FUNCTION_BLOCK pidCtl (* Composite Function Block Type *)
  (* Standard: 61499-2 *)
  (* Version 1.0.1, 11/15/2023, ApplicationLibDevTeam, Schneider Electric, First Version *)
  PACKAGE Hidryco.HidrycoLib;
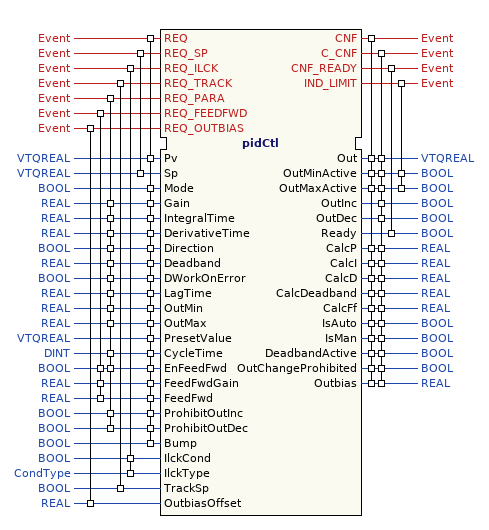
  EVENT_INPUT
    REQ WITH Pv, Gain, DerivativeTime, IntegralTime, Direction, Deadband, DWorkOnError, Mode, PresetValue, CycleTime, EnFeedFwd, FeedFwdGain, FeedFwd, LagTime, OutMin, OutMax, ProhibitOutInc, ProhibitOutDec, Bump; (* Request to execute PID in auto or manual mode *)
    REQ_SP WITH Sp; (* Request for setpoint execution *)
    REQ_ILCK WITH IlckCond, IlckType; (* Request to update interlock *)
    REQ_TRACK WITH TrackSp; (* Request for track setpoint *)
    REQ_PARA WITH Gain, DerivativeTime, IntegralTime, Direction, Deadband, DWorkOnError, CycleTime, EnFeedFwd, LagTime, OutMin, OutMax, ProhibitOutInc, ProhibitOutDec; (* Request for parameter updates *)
    REQ_FEEDFWD WITH FeedFwd, EnFeedFwd, FeedFwdGain; (* Request for executing feedforward gain *)
    REQ_OUTBIAS WITH OutbiasOffset; (* Request to update outbias offset value *)
  END_EVENT
  EVENT_OUTPUT
    CNF WITH Out, OutMinActive, OutMaxActive, CalcP, CalcI, CalcD, CalcDeadband, CalcFf, IsAuto, IsMan, DeadbandActive, OutChangeProhibited, Outbias; (* Execution confirmation *)
    C_CNF WITH Out, OutMinActive, OutMaxActive, OutInc, OutDec, CalcP, CalcI, CalcD, CalcDeadband, CalcFf, IsAuto, IsMan, DeadbandActive, OutChangeProhibited, Outbias; (* Cyclic execution confirmation *)
    CNF_READY WITH Ready; (* Execution confirmation of control module ready *)
    IND_LIMIT WITH OutMinActive, OutMaxActive; (* Indication for output low/high limit activated *)
  END_EVENT
  VAR_INPUT
    Pv : VTQREAL; (* Process value *)
    Sp : VTQREAL; (* Setpoint *)
    Mode : BOOL; (* 1 = Auto, 0 = Manual mode *)
    Gain : REAL; (* Gain parameter for PID calculation *)
    IntegralTime : REAL; (* Integral parameter for I calculation *)
    DerivativeTime : REAL; (* Derivative parameter for D calculation *)
    Direction : BOOL := FALSE; (* Direction for error calculation (0 = PV-SP; 1 = SP-PV) *)
    Deadband : REAL; (* Deadband for I and D calculation *)
    DWorkOnError : BOOL; (* 1 = Derivative applied to error; 0 = Derivative applied to Pv *)
    LagTime : REAL; (* Lag time parameter for D calculation *)
    OutMin : REAL; (* Minimal output value *)
    OutMax : REAL; (* Maximal output value *)
    PresetValue : VTQREAL; (* Preset value for Out *)
    CycleTime : DINT; (* Timebase for PID calculation (ms) *)
    EnFeedFwd : BOOL; (* 1 = Feed forward usage active *)
    FeedFwdGain : REAL; (* Feed forward Gain parameter *)
    FeedFwd : REAL; (* Feedforward *)
    ProhibitOutInc : BOOL; (* 1 = Output increment prohibited *)
    ProhibitOutDec : BOOL; (* 1 = Output decrement prohibited *)
    Bump : BOOL; (* 1 =Transition to automatic mode with bump ,0= Bumpless transition to automatic mode *)
    IlckCond : BOOL; (* 1 = Interlock condition active *)
    IlckType : CondType; (* Type of condition interlock, (0 = Normal, 1 = Process interlock/Sequence interlock) *)
    TrackSp : BOOL; (* 1 = Track setpoint *)
    OutbiasOffset : REAL; (* Output offset (bias), calculated based on integral component *)
  END_VAR
  VAR_OUTPUT
    Out : VTQREAL; (* Calculated Output value *)
    OutMinActive : BOOL; (* 1 = Out has reached OutMinLimit *)
    OutMaxActive : BOOL; (* 1 = Out has reached OutMaxLimit *)
    OutInc : BOOL; (* 1 = Output is increasing *)
    OutDec : BOOL; (* 1 = Output is decreasing *)
    Ready : BOOL; (* 1 = Control module ready for operation *)
    CalcP : REAL; (* Calculated proportional part *)
    CalcI : REAL; (* Calculated intergral part *)
    CalcD : REAL; (* Calculated derivative part *)
    CalcDeadband : REAL; (* Calculated Deadband *)
    CalcFf : REAL; (* Calculated Feed forward value *)
    IsAuto : BOOL; (* 1 = Automatic mode detected *)
    IsMan : BOOL; (* 1 = Manual mode detected *)
    DeadbandActive : BOOL; (* 1 = Deadband mode is active *)
    OutChangeProhibited : BOOL; (* 1 = Output changed prohibited *)
    Outbias : REAL; (* Output offset (bias) value in Auto Mode and Integration time is zero *)
  END_VAR
  (* Event to bing the FF value in the FB Will wait the normal cycle to be applyed. Event not connected in purpose *)
  (* PID Calculation *)
  FBS
    cycleEvent : E_CYCLE;
    pidSC : pidSC;
  END_FBS
  EVENT_CONNECTIONS
    cycleEvent.EO TO pidSC.C_REQ;
    pidSC.CNF TO CNF;
    pidSC.C_CNF TO C_CNF;
    pidSC.IND_LIMIT TO IND_LIMIT;
    REQ_PARA TO pidSC.OP_PARA;
    pidSC.CNF_READY TO CNF_READY;
    REQ_ILCK TO pidSC.REQ_ILCK;
    REQ_TRACK TO pidSC.REQ_TRACK;
    REQ_OUTBIAS TO pidSC.REQ_OUTBIAS;
    REQ TO pidSC.REQ;
    pidSC.C_START TO cycleEvent.START;
    pidSC.C_STOP TO cycleEvent.STOP;
    REQ_SP TO pidSC.REQ;
  END_CONNECTIONS
  DATA_CONNECTIONS
    FeedFwd TO pidSC.FeedFwd;
    Sp TO pidSC.Sp;
    EnFeedFwd TO pidSC.FeedFwdOn;
    FeedFwdGain TO pidSC.FeedFwdGain;
    ProhibitOutInc TO pidSC.ProhibitOutInc;
    ProhibitOutDec TO pidSC.ProhibitOutDec;
    Pv TO pidSC.Pv;
    Gain TO pidSC.Gain;
    DerivativeTime TO pidSC.Rate;
    IntegralTime TO pidSC.Reset;
    LagTime TO pidSC.LagTime;
    OutMin TO pidSC.OutMinLimit;
    OutMax TO pidSC.OutMaxLimit;
    PresetValue TO pidSC.PresetValue;
    Deadband TO pidSC.Deadband;
    Direction TO pidSC.Direction;
    DWorkOnError TO pidSC.DWorkOnError;
    pidSC.Out TO Out;
    pidSC.OutMinActive TO OutMinActive;
    pidSC.OutMaxActive TO OutMaxActive;
    pidSC.OutInc TO OutInc;
    pidSC.OutDec TO OutDec;
    pidSC.CalcP TO CalcP;
    pidSC.CalcI TO CalcI;
    pidSC.CalcD TO CalcD;
    pidSC.CalcDeadband TO CalcDeadband;
    pidSC.CalcFf TO CalcFf;
    pidSC.IsAuto TO IsAuto;
    pidSC.IsMan TO IsMan;
    pidSC.DeadbandActive TO DeadbandActive;
    pidSC.OutChangeProhibited TO OutChangeProhibited;
    Mode TO pidSC.Mode;
    pidSC.Outbias TO Outbias;
    Bump TO pidSC.Bump;
    OutbiasOffset TO pidSC.OutbiasOffset;
    CycleTime TO pidSC.TimeBase;
    pidSC.Ready TO Ready;
    IlckCond TO pidSC.IlckCond;
    IlckType TO pidSC.IlckType;
    TrackSp TO pidSC.TrackSp;
    pidSC.TimeOut TO cycleEvent.DT;
  END_CONNECTIONS
END_FUNCTION_BLOCK
